// TwinCAT 3 PLC project TcLog
// Title: TcLog
// Company: Benedikt Geisler
// Author: Benedikt Geisler
// ProjectVersion: 0.6.1
// Description: TcLog provides logging functionality to TwinCAT.
// ProgramVersion: 3.1.4026.12
// libraries:
//   Base Interfaces,newest,System
//   Tc2_Standard, * (Beckhoff Automation GmbH)
//   Tc2_System, * (Beckhoff Automation GmbH)
//   Tc2_Utilities, * (Beckhoff Automation GmbH)
//   Tc3_DynamicMemory, * (Beckhoff Automation GmbH)
//   Tc3_Module, * (Beckhoff Automation GmbH)
//   TcUnit, * (www.tcunit.org)
// project tree:
//   / Constants.TcGVL
//   Logger/ LogLevelToAdsLogMsgType.TcPOU, TcLog.TcPOU, TcLogCore.TcPOU, TcLogTrig.TcPOU
//   Logger/_Tests/ TestWrapper_NET.TcPOU
//   StringBuilder/_Interfaces/ ILimitedStringBuilder.TcIO, IStringBuilder.TcIO
//   Utils/ AnyToString.TcPOU, DateTime.TcPOU, DeleteOldFiles.TcPOU, DynamicStringBuffer.TcPOU, GetFileAgeInSeconds.TcPOU
//   Utils/_DataTypes/ DeleteFilesState.TcDUT, PersistToFileState.TcDUT
//   Logger/_DataTypes/ ErrorCodes.TcDUT, LogLevels.TcDUT, RollingIntervals.TcDUT, Error.TcDUT, LoggingConfiguration.TcDUT
//   Logger/_Interfaces/ ILog.TcIO, ILogCore.TcIO
//   StringBuilder/ StringBuilder.TcPOU
//   Utils/_Tests/ ConvertAnyToString_TEST.TcPOU, DateTime_TEST.TcPOU, DynamicStringBuffer_TEST.TcPOU
// real-time tasks:
//   TASK PlcTask1: cycle T#10ms, priority 21, ADS port 351

// ---- Utils/_DataTypes/DeleteFilesState.TcDUT
// States for state machine used in `DeleteOldFiles`.
{attribute 'qualified_only'}
{attribute 'strict'}
TYPE INTERNAL DeleteFilesState :
(
	Idle := 0,
  SearchNextFile,
  WaitUntilExecutionDone,
  ProcessFoundFiles,
  CheckIfFileIsDirectory,
  CheckFileTime,
  DeleteFile,
  FileDeleted
);
END_TYPE

// ---- Utils/_DataTypes/PersistToFileState.TcDUT
// States for state machine used in `DynamicStringBuffer.PersistToFile`
{attribute 'qualified_only'}
{attribute 'strict'}
TYPE INTERNAL PersistToFileState :
(
	Idle := 0,
  OpenFile,
  GetStringFromFifo,
  AppendDataToFile,
  CloseFile
);
END_TYPE

// ---- Logger/_DataTypes/ErrorCodes.TcDUT
/// Provides error codes for TcLogCore
{attribute 'qualified_only'}
{attribute 'strict'}
{attribute 'to_string'}
TYPE ErrorCodes : 
(
	None := 0,
	OpeningFileFailed,
	WritingToFileFailed,
	ClosingFileFailed,
	EnumeratingFilesInSpecifiedDirectoryFailed,
	DeletingFileFailed,
	FifoOverflow
);
END_TYPE

// ---- Logger/_DataTypes/LogLevels.TcDUT
/// Log level of message to be logged.
{attribute 'qualified_only'}
{attribute 'strict'}
{attribute 'to_string'}
TYPE LogLevels :
(
	Debug := 0,
	Information,
	Warning,
	Error,
	Fatal
);
END_TYPE

// ---- Logger/_DataTypes/RollingIntervals.TcDUT
/// Rolling interval to create a new log file when expired. 
{attribute 'qualified_only'}
{attribute 'strict'}
{attrivute 'to_string'}
TYPE RollingIntervals :
(
	None := 0,
	Hourly,
	Daily,
	Monthly
);
END_TYPE

// ---- Logger/_DataTypes/Error.TcDUT
/// This is the error type used in this library.
TYPE Error :
STRUCT
  /// `TRUE` signals an active error
	Active : BOOL;
  /// Error code of type `ErrorCodes`
	Code : INT;
  /// Plain text error message
	Info : Tc2_System.T_MaxString;
END_STRUCT
END_TYPE

// ---- Logger/_DataTypes/LoggingConfiguration.TcDUT
/// Configuration of TcLogCore
TYPE LoggingConfiguration :
STRUCT
  /// File name where the logs should be written to. Should not include path.
	FileName : Tc2_System.T_MaxString;
  /// File path where the logs should be written to. Will be prefixed to `FileName`
	FilePath : Tc2_System.T_MaxString;
  /// Whether to include the instance path of TcLog into the log message or not.
	IncludeInstancePath : BOOL;
  /// Whether to write the logs to ADS output or not.
	WriteToAds : BOOL;
  /// Rolling interval: when to create a new log file.
	RollingInterval : RollingIntervals;
  /// What is the minimum log level that gets logged?
	MinimumLevel : LogLevels;
  /// Which delimiter should be used between the different parts of the log string?
	Delimiter : STRING(1);
  /// When should old log files be deleted? Unit: days. Set it to `0` if log files should never be deleted. 
	LogFileLifespan : UINT;
  /// Format of timestamp. See `TcLogCore.TimestampFormat` for formatting options.
	TimestampFormat : STRING;
  /// Log only valid timestamps (skip log messages during time initialization (first few cycles)
  	ValidTimestampsOnly: BOOL;
END_STRUCT
END_TYPE

// ---- Constants.TcGVL
{attribute 'qualified_only'}
VAR_GLOBAL CONSTANT
  /// Fifo overhead needed to manage the string buffer
  FifoOverhead : UDINT := 10;
  /// Buffer size of temporary buffer used to persist all log messages in one cycle. 
	BufferSize : UDINT := (100 * (Tc2_System.MAX_STRING_LENGTH + FifoOverhead));
END_VAR

// ---- StringBuilder/_Interfaces/ILimitedStringBuilder.TcIO
{attribute 'hide'}
INTERFACE INTERNAL ILimitedStringBuilder

METHOD Append : IStringBuilder // Append text TO t current build STRING.
VAR_INPUT
    Text : Tc2_System.T_MaxString; //Text to append to current build string
END_VAR
END_METHOD

METHOD AppendIf : IStringBuilder
VAR_INPUT
    Condition : BOOL;
    Text : Tc2_System.T_MaxString;
END_VAR
END_METHOD

METHOD Reset : ILimitedStringBuilder //Reset current build STRING TO an empty STRING.
END_METHOD

METHOD ToString : Tc2_System.T_MaxString //Returns current build STRING.
END_METHOD

END_INTERFACE

// ---- StringBuilder/_Interfaces/IStringBuilder.TcIO
{attribute 'hide'}
INTERFACE INTERNAL IStringBuilder

METHOD Append : IStringBuilder // Append text TO t current build STRING.
VAR_INPUT
    Text : Tc2_System.T_MaxString; //Text to append to current build string
END_VAR
END_METHOD

METHOD AppendIf : IStringBuilder
VAR_INPUT
    Condition : BOOL;
    Text : Tc2_System.T_MaxString;
END_VAR
END_METHOD

METHOD InsertAtLocation : IStringBuilder
VAR_INPUT
    Text : Tc2_System.T_MaxString;
    Position : INT;
END_VAR
END_METHOD

METHOD PadLeft : IStringBuilder
VAR_INPUT
    text : Tc2_System.T_MaxString; // Text to append to current build string
    length : INT; // Total length of text + padding
    c : STRING(1); // Character to be padded left of text
END_VAR
END_METHOD

METHOD Reset : ILimitedStringBuilder //Reset current build STRING TO an empty STRING.
END_METHOD

METHOD ToString : Tc2_System.T_MaxString //Returns current build STRING.
END_METHOD

END_INTERFACE

// ---- Logger/_Interfaces/ILog.TcIO
INTERFACE ILog

METHOD SetLogger : BOOL
VAR_INPUT
    ref2Core : ILogCore;
END_VAR
END_METHOD

END_INTERFACE

// ---- Logger/_Interfaces/ILogCore.TcIO
INTERFACE ILogCore EXTENDS __System.IQueryInterface

// Logger method.
// Logs data in custom format. No additional formatting will be done.
METHOD LogCustomFormat : BOOL
VAR_INPUT
    data : Tc2_System.T_MaxString; // Data to be logged. No additional formatting will be done.
END_VAR
END_METHOD

// Logger method.
// Logs in the standard format. This includes
// - timestamp
// - log level
// - log message
// - instance path of logging source (optional)
// The message will only be logged if the logging level exceeds the configured minimum logging level.
METHOD LogStandardFormat : BOOL
VAR_INPUT
    data : Tc2_System.T_MaxString; // Data to be logged. Additional formatting wil be done.
    instancePath : Tc2_System.T_MaxString; // Instance path of calling logger to locate source of logging message.
    logLevel : LogLevels; // Log level of message.
END_VAR
END_METHOD

END_INTERFACE

// ---- Logger/LogLevelToAdsLogMsgType.TcPOU
// Converts TcLog.LogLevels into Tc2_System.ADSLOG_MSGTYPEs.
{attribute 'hide'}
FUNCTION INTERNAL LogLevelToAdsLogMsgType : DWORD
VAR_INPUT
  logLevel : LogLevels;
END_VAR
VAR
  _retVal : DWORD;
END_VAR

CASE logLevel OF
  LogLevels.Debug, LogLevels.Information:
    _retVal := Tc2_System.ADSLOG_MSGTYPE_HINT;
  LogLevels.Warning:
    _retVal := Tc2_System.ADSLOG_MSGTYPE_WARN;
  LogLevels.Error, LogLevels.Fatal:
    _retVal := Tc2_System.ADSLOG_MSGTYPE_ERROR;
  ELSE
    _retVal := Tc2_System.ADSLOG_MSGTYPE_HINT;
END_CASE

LogLevelToAdsLogMsgType := _retVal;

END_FUNCTION

// ---- Logger/TcLog.TcPOU
/// `TcLog` is the client side of the logger.  
///
/// It is used to send the logs to `TcLogCore`. Typically, it is instantiated
/// once in each `FUNCTION_BLOCK` or `PROGRAM` where logging is done. The same 
/// instance can then be used for all logging within that POU. 
///
/// `TcLog` implements a string builder that facilitates the compilation of the log
/// message without the need for external data type conversions or multiple chained `CONCAT` calls.
/// See the method section for more information.
///
/// The last method to call after the log message has been built is one of ´[Debug|Information|Warning|Error|Fatal]`. 
/// This sets the log level of the message and sends it off to the log message queue of `TcLogCore` where it will
/// be processed according to its configuration.
{attribute 'hide_all_locals'}
{attribute 'reflection'} 
FUNCTION_BLOCK TcLog IMPLEMENTS ILog
VAR
  _logConditionSatisfied : BOOL; // flag that indicates, whether log condition has been satisfied.
                                // Logging will only be carried out it this evaluates to TRUE.                    
  _logDataInitialized : BOOL; // flag that indicate, whether log data has been initialized.
                             // Necessary for configuration methods to provide a fluent interface.                            
  _logData : Tc2_System.T_MaxString; // contains message to be logged.
  _usedLogger : ILogCore;
  {attribute 'instance-path'} 
  {attribute 'noinit'} 
  _instancePath : STRING; // contains instance path
END_VAR
VAR_STAT
  {attribute 'hide'}
  s_loggerSingletonInstance : ILogCore; // Wires up TcLog ("Client") to TcLogCore ("Server") (Singleton-Behaviour)
END_VAR
VAR CONSTANT
  InvalidLoggerReference : UDINT := 0;
END_VAR

/// Appends any given data to the log string. The type of the provided data
/// has to be one of the [standard data types](https://infosys.beckhoff.com/english.php?content=../content/1033/tc3_plc_intro/2529388939.html&id=).
/// This method can be chained.
METHOD AppendAny : REFERENCE TO TcLog
VAR_INPUT
  /// data to be appended to log string.
  data : ANY;
END_VAR
InitializeLogData();

_logData := Tc2_Standard.CONCAT(_logData, AnyToString(data));

AppendAny REF= THIS^;
END_METHOD

/// Appends another string to the log message.
/// This method can be chained.
METHOD AppendString : REFERENCE TO TcLog
VAR_INPUT
  /// data to be appended to log string.
  data : Tc2_System.T_MaxString; 
END_VAR
InitializeLogData();

_logData := Tc2_Standard.CONCAT(_logData, data);
  
AppendString REF= THIS^;
END_METHOD

/// Appends information about the given variable to the log string. 
/// This method can be chained.
/// Example: 

/// ```st
/// VAR
///   Logger: TcLog;
///    myInt : INT := 10;
///   myVarInfo : __SYSTEM.VAR_INFO := __VARINFO(myInt);
/// END_VAR
/// Logger.AppendVariable(myVarInfo, myInt);
/// ```
///
METHOD AppendVariable : REFERENCE TO TcLog
VAR_INPUT
  /// [VAR_INFO](https://infosys.beckhoff.com/index.php?content=../content/1031/tc3_plc_intro/3527777675.html&id=) of variable to be appended to log string.
  varInfo : __SYSTEM.VAR_INFO;
  /// Value of variable to be appended to log string.
  value : ANY; 
END_VAR
VAR
  format : Tc2_Utilities.FB_FormatString;
  symbolName : Tc2_System.T_MaxString;
  typeName : Tc2_System.T_MaxString;
END_VAR
InitializeLogData();

symbolName := varInfo.Symbol;
typeName := varInfo.TypeName; 

format(
  sFormat := '%s [%s] : ',
  arg1 := Tc2_Utilities.F_STRING(symbolName),
  arg2 := Tc2_Utilities.F_STRING(typeName));
  
AppendString(format.sOut);
AppendAny(value);

AppendVariable REF= THIS^;
END_METHOD

/// Logs the log string in DEBUG level.
METHOD Debug : BOOL
VAR_INPUT
  /// Message to be appended to log string.
  message : Tc2_System.T_MaxString; 
END_VAR
InitializeLogData();
IF _logConditionSatisfied THEN
  IF _usedLogger <> InvalidLoggerReference THEN 
    _usedLogger.LogStandardFormat(Tc2_Standard.CONCAT(_logData, message), ShortenInstancePath(_instancePath), LogLevels.Debug); 
  ELSE
    Tc2_System.ADSLOGSTR(ADSLOG_MSGTYPE_LOG OR LogLevelToAdsLogMsgType(LogLevels.Error), 'usedLogger: No valid reference', ''); 
  END_IF
END_IF
_logDataInitialized := FALSE;
END_METHOD

/// Logs the log string in ERROR level.
METHOD Error : BOOL
VAR_INPUT
  /// Message to be appended to log string.
  message : Tc2_System.T_MaxString; 
END_VAR
InitializeLogData();
IF _logConditionSatisfied THEN
  IF _usedLogger <> InvalidLoggerReference THEN 
    _usedLogger.LogStandardFormat(Tc2_Standard.CONCAT(_logData, message), ShortenInstancePath(_instancePath), LogLevels.Error); 
  ELSE
    Tc2_System.ADSLOGSTR(ADSLOG_MSGTYPE_LOG OR LogLevelToAdsLogMsgType(LogLevels.Error), 'usedLogger: No valid reference', ''); 
  END_IF
END_IF
_logDataInitialized := FALSE;
END_METHOD

/// Logs the log string in FATAL level.
METHOD Fatal : BOOL
VAR_INPUT
  /// Message to be appended to log string.
  message : Tc2_System.T_MaxString; 
END_VAR
InitializeLogData();
IF _logConditionSatisfied THEN
  IF _usedLogger <> InvalidLoggerReference THEN 
    _usedLogger.LogStandardFormat(Tc2_Standard.CONCAT(_logData, message), ShortenInstancePath(_instancePath), LogLevels.Fatal); 
  ELSE
    Tc2_System.ADSLOGSTR(ADSLOG_MSGTYPE_LOG OR LogLevelToAdsLogMsgType(LogLevels.Error), 'usedLogger: No valid reference', ''); 
  END_IF
END_IF
_logDataInitialized := FALSE;
END_METHOD

/// Logs the log string in INFORMATION level.
METHOD Information : BOOL
VAR_INPUT
  /// Message to be appended to log string.
  message : Tc2_System.T_MaxString; 
END_VAR
InitializeLogData();
IF _logConditionSatisfied THEN
  IF _usedLogger <> InvalidLoggerReference THEN 
    _usedLogger.LogStandardFormat(Tc2_Standard.CONCAT(_logData, message), ShortenInstancePath(_instancePath), LogLevels.Information); 
  ELSE
    Tc2_System.ADSLOGSTR(ADSLOG_MSGTYPE_LOG OR LogLevelToAdsLogMsgType(LogLevels.Error), 'usedLogger: No valid reference', ''); 
  END_IF
END_IF
_logDataInitialized := FALSE;
END_METHOD

/// Initializes the reference to the core logger. Should only be called once from the core logger directly.
METHOD PUBLIC Init : BOOL
VAR_INPUT
  /// Reference to TcLoggerCore instance.
  ref2Core : ILogCore; 
END_VAR
IF s_loggerSingletonInstance = 0 THEN
	s_loggerSingletonInstance := ref2Core;
END_IF
END_METHOD

// Necessary to provide a fluent interface of the function. 
// Has to be called at the begin of any method that returns a reference to THIS^
METHOD PRIVATE InitializeLogData : BOOL
IF NOT _logDataInitialized THEN
  _logConditionSatisfied := TRUE;
  _logData := '';
  _logDataInitialized := TRUE;
  IF _usedLogger = 0 THEN _usedLogger := s_loggerSingletonInstance; END_IF
END_IF
END_METHOD

/// Conditional execution of the log command. Only executes logging when Cond = TRUE.
METHOD OnCondition : REFERENCE TO TcLog
VAR_INPUT
  /// Logs data only if this condition evaluates to TRUE.
  cond : BOOL; 
END_VAR
InitializeLogData();

_logConditionSatisfied := cond;

OnCondition REF= THIS^;
END_METHOD

/// Initializes the reference to the core logger. This enables you to use several
/// loggers with different configurations in one project.
METHOD SetLogger : BOOL
VAR_INPUT
  /// Reference to Core Logger
  ref2Core : ILogCore; 
END_VAR
_usedLogger := ref2Core;
END_METHOD

// Helper method. Shortens the instance path by omitting superfluent information
// such as concrete logger instance and plc/project names.
{attribute 'hide'}
METHOD PRIVATE ShortenInstancePath : Tc2_System.T_MaxString
VAR_INPUT
  path : Tc2_System.T_MaxString; // Instance path to be shortened.
END_VAR
VAR
  i : UINT;
  shortenedPath : Tc2_System.T_MaxString;
  positionInString : INT := 0;
  positionOfLastDot : INT := 0;
END_VAR
shortenedPath := path;

// Find last '.'
WHILE(Tc2_Standard.FIND(shortenedPath, '.') > 0) DO
  positionInString := Tc2_Standard.FIND(shortenedPath, '.');
  shortenedPath := Tc2_Standard.DELETE(shortenedPath, positionInString+1, 0); 
  positionOfLastDot := positionOfLastDot+positionInString;
END_WHILE

shortenedPath := Path;
// Delete instantiation of this FB (obvious information)
shortenedPath := Tc2_Standard.DELETE(shortenedPath, Tc2_Standard.LEN(shortenedPath)-positionOfLastDot+1, positionOfLastDot);
// Delete project information
positionInString := Tc2_Standard.FIND(shortenedPath, '.');
shortenedPath := Tc2_Standard.DELETE(shortenedPath, positionInString+1, 0);
// Delete PLC information
positionInString := Tc2_Standard.FIND(shortenedPath, '.');
shortenedPath := Tc2_Standard.DELETE(shortenedPath, positionInString+1, 0);

ShortenInstancePath := shortenedPath;
END_METHOD

/// Logs directly to ADS log, ignoring the settings of the base logger.
METHOD ToAdsLog : BOOL
VAR_INPUT
  /// Log level in which message should be logged to ADS.
  logLevel : LogLevels; 
END_VAR
InitializeLogData();

IF _logConditionSatisfied THEN
  Tc2_System.ADSLOGSTR(ADSLOG_MSGTYPE_LOG OR LogLevelToAdsLogMsgType(logLevel), _logData, ''); 
END_IF

_logDataInitialized := FALSE;
END_METHOD

/// Saves custom formatted log string. 
/// No addtitional information will be added, no formatting will be applied.
METHOD ToCustomFormat : BOOL
VAR_INPUT
  /// Message to be appended to log string.
  message : Tc2_System.T_MaxString; 
END_VAR
InitializeLogData();
IF _logConditionSatisfied THEN
  IF _usedLogger <> InvalidLoggerReference THEN 
    _usedLogger.LogCustomFormat(Tc2_Standard.CONCAT(_logData, message)); 
  ELSE
    Tc2_System.ADSLOGSTR(ADSLOG_MSGTYPE_LOG OR LogLevelToAdsLogMsgType(LogLevels.Error), 'usedLogger: No valid reference', ''); 
  END_IF
END_IF
_logDataInitialized := FALSE;
END_METHOD

/// Logs the log string in WARNING level.
METHOD Warning : BOOL
VAR_INPUT
  /// Message to be appended to log string.
  message : Tc2_System.T_MaxString; 
END_VAR
InitializeLogData();
IF _logConditionSatisfied THEN
  IF _usedLogger <> InvalidLoggerReference THEN 
    _usedLogger.LogStandardFormat(Tc2_Standard.CONCAT(_logData, message), ShortenInstancePath(_instancePath), LogLevels.Warning); 
  ELSE
    Tc2_System.ADSLOGSTR(ADSLOG_MSGTYPE_LOG OR LogLevelToAdsLogMsgType(LogLevels.Error), 'usedLogger: No valid reference', ''); 
  END_IF
END_IF
_logDataInitialized := FALSE;
END_METHOD

END_FUNCTION_BLOCK

// ---- Utils/AnyToString.TcPOU
/// Converts value of input data to string, where the input type can be any of 
/// the standard data types.
FUNCTION AnyToString : Tc2_System.T_MaxString
VAR_INPUT
  /// Input data
  data : ANY;
END_VAR
VAR
  _anyByte : POINTER TO BYTE;
  _anyUSINT : POINTER TO USINT;
  _anyInt : POINTER TO INT;
  _anyUInt : POINTER TO UINT;
  _anyUDInt : POINTER TO UDINT;
  _anySInt : POINTER TO SINT;
  _anyDInt : POINTER TO DINT;
  _anyLInt : POINTER TO LINT;
  _anyULInt : POINTER TO ULINT;
  _anyWord : POINTER TO WORD;
  _anyLWord : POINTER TO LWORD;
  _anyReal : POINTER TO REAL;
  _anyLReal : POINTER TO LREAL;
  _anyDateAndTime : POINTER TO DATE_AND_TIME;
  _anyDate : POINTER TO DATE;
  _anyTime : POINTER TO TIME;
  _anyWString : POINTER TO WSTRING;
  _anyTOD : POINTER TO TOD;
  _anyString : POINTER TO STRING;
  _string : T_MAXSTRING;
  _wString : WSTRING;
END_VAR

IF data.TypeClass = __SYSTEM.TYPE_CLASS.TYPE_BYTE THEN
  _anyByte := data.pValue;
  AnyToString := BYTE_TO_STRING(_anyByte^);
    
ELSIF data.TypeClass = __SYSTEM.TYPE_CLASS.TYPE_INT THEN
  _anyInt := data.pValue;
  AnyToString := INT_TO_STRING(_anyInt^);
    
ELSIF data.TypeClass = __SYSTEM.TYPE_CLASS.TYPE_UINT THEN
  _anyUInt := data.pValue;
  AnyToString := UINT_TO_STRING(_anyUInt^);
    
ELSIF data.TypeClass = __SYSTEM.TYPE_CLASS.TYPE_UDINT THEN
  _anyUDInt := data.pValue;
  AnyToString := UDINT_TO_STRING(_anyUDInt^);
    
ELSIF data.TypeClass = __SYSTEM.TYPE_CLASS.TYPE_SINT THEN
  _anySInt := data.pValue;
  AnyToString := SINT_TO_STRING(_anySInt^);
    
ELSIF data.TypeClass = __SYSTEM.TYPE_CLASS.TYPE_USINT THEN
  _anyUSInt := data.pValue;
  AnyToString := USINT_TO_STRING(_anyUSInt^);
    
ELSIF data.TypeClass = __SYSTEM.TYPE_CLASS.TYPE_DINT THEN
  _anyDInt := data.pValue;
  AnyToString := DINT_TO_STRING(_anyDInt^);
    
ELSIF data.TypeClass = __SYSTEM.TYPE_CLASS.TYPE_LINT THEN
  _anyLInt := data.pValue;
  AnyToString := LINT_TO_STRING(_anyLInt^);
      
ELSIF data.TypeClass = __SYSTEM.TYPE_CLASS.TYPE_ULINT THEN
  _anyULInt := data.pValue;
  AnyToString := ULINT_TO_STRING(_anyULInt^);
  
ELSIF data.TypeClass = __SYSTEM.TYPE_CLASS.TYPE_WORD THEN
  _anyWord := data.pValue;
  AnyToString := WORD_TO_STRING(_anyWord^);
    
ELSIF data.TypeClass = __SYSTEM.TYPE_CLASS.TYPE_LWORD THEN
  _anyLWord := data.pValue;
  AnyToString := LWORD_TO_STRING(_anyLWord^);
  
ELSIF data.TypeClass = __SYSTEM.TYPE_CLASS.TYPE_REAL THEN
  _anyReal := data.pValue;
  AnyToString := REAL_TO_STRING(_anyReal^);
  
ELSIF data.TypeClass = __SYSTEM.TYPE_CLASS.TYPE_LREAL THEN
  _anyLReal := data.pValue;
  AnyToString := LREAL_TO_STRING(_anyLReal^);
  
ELSIF data.TypeClass = __SYSTEM.TYPE_CLASS.TYPE_DATEANDTIME THEN
  _anyDateAndTime := data.pValue;
  AnyToString := DT_TO_STRING(_anyDateAndTime^);  
  
ELSIF data.TypeClass = __SYSTEM.TYPE_CLASS.TYPE_DATE THEN
  _anyDate := data.pValue;
  AnyToString := DATE_TO_STRING(_anyDate^);
  
ELSIF data.TypeClass = __SYSTEM.TYPE_CLASS.TYPE_TIME THEN
  _anyTime := data.pValue;
  AnyToString := TIME_TO_STRING(_anyTime^);
  
ELSIF data.TypeClass = __SYSTEM.TYPE_CLASS.TYPE_STRING THEN
  _anyString := data.pValue;
  AnyToString := _anyString^;
  
ELSIF data.TypeClass = __SYSTEM.TYPE_CLASS.TYPE_WSTRING THEN
  _anyWString := data.pValue;
  _wString := _anyWString^;
  Tc2_Utilities.WSTRING_TO_STRING2(ADR(_string), ADR(_wString), SIZEOF(_wString));
  AnyToString := _string;
  
ELSIF data.TypeClass = __SYSTEM.TYPE_CLASS.TYPE_TIMEOFDAY THEN
  _anyTOD := data.pValue;
  AnyToString := TOD_TO_STRING(_anyTOD^);
  
ELSE
  AnyToString := TO_STRING(data.pValue^);
END_IF

END_FUNCTION

// ---- Logger/TcLogCore.TcPOU
/// `TcLogCore` provides the base functionality of the logger and sets the configuration.
/// The logger can be configured by calling its methods that set the configuration.
///
/// > [!NOTE]
/// > `TcLogCore.RunLogger()` should be called once each cycle. The configuration methods should be called **before** 
/// > `RunLogger` is called.
///
/// When declaring an instance of TcLogCore, the ininital buffer size has to be set. If the buffer size is set too low, it will expand
/// automatically if enough memory is available.
///
/// To set the inital buffer size to accomodate 100 messages, use it like this:
///
/// ```st
/// VAR
///   myLogger: TcLogCore(BufferSize := 100 * (Tc2_System.MAX_STRING_LENGTH * Constants.FifoOverhead));
/// END_VAR
/// ```
///
{attribute 'hide_all_locals'}
FUNCTION_BLOCK TcLogCore IMPLEMENTS ILogCore
VAR
	_loggingSingleton : TcLog; // Logger-Singleton: Required to provide Singleton-functionality for TcLog.
	_utcTimeAsFileTime : Tc2_Utilities.T_FILETIME; // Current utc time as filetime
	_localTimeAsSystemTime : Tc2_Utilities.TIMESTRUCT; // Current local time as timestring
	_localTimeAsString : STRING; // Current local time as string
	_logCache : DynamicStringBuffer; // Dynamic string buffer to cache logs to be processed
	_startLoggingConfiguration : BOOL; // Aux variable to provide fluent interface.
	_internalErrorOccured : BOOL; // Aux variable to log internal errors to Error-property.                                                   				
	_config : LoggingConfiguration; // Logging configuration. Is set by invoking configuration methods.
	_error : Error; // Contains information about internal error.
	_busy : BOOL; // Logger is busy, typically with writing logs to the file system.
  _timeInfoReady : BOOL := FALSE; // Set to true once the time information is available
END_VAR

// Nothing to be done here. Logger works by invoking its methods.
// "RunLogger" contains all the implementation that has to be processed cyclically.

// Builds logging configuration.
// Required to provide a fluent interface.
// Has to be called at the begin of each method that configures the logger.
{attribute 'hide'}
METHOD PRIVATE BuildLoggingConfiguration : BOOL
IF NOT _startLoggingConfiguration THEN
	_startLoggingConfiguration := TRUE;
	
	_config.RollingInterval := RollingIntervals.Daily;
	_config.WriteToAds := FALSE;
	_config.FileName := '';
	_config.FilePath := 'c:\';
	_config.MinimumLevel := LogLevels.Debug;
	_config.Delimiter := '|';
	_config.IncludeInstancePath := FALSE;
	_config.LogFileLifespan := 0;
	_config.TimestampFormat := 'YYYYMMDD_hhmm_';
	_config.ValidTimestampsOnly := FALSE;
END_IF
END_METHOD

/// `Busy` evaluates to `TRUE` as long as the log file is kept open to append new log messages
/// or there are pending messages in the queue to be written to the logfile.
{attribute 'monitoring':='call'}
PROPERTY Busy : BOOL
GET
Busy := _busy;
END_GET
SET // PRIVATE
_busy := Busy;
END_SET
END_PROPERTY

/// Returns the current configuration of the logger.
{attribute 'monitoring':='variable'}
PROPERTY Configuration : LoggingConfiguration
GET
Configuration := _config;
END_GET
END_PROPERTY

/// Configuration method which sets the lifespan of log files. Once exceeded, they will be deleted.
METHOD DeleteLogFilesAfterDays : REFERENCE TO TcLogCore
VAR_INPUT
  /// Lifespan of logfiles in days.
	lifespan : UINT; 
END_VAR
BuildLoggingConfiguration();

_config.LogFileLifespan := lifespan;

DeleteLogFilesAfterDays REF= THIS^;
END_METHOD

/// Returns information about internal errors.
{attribute 'monitoring':='call'}
PROPERTY Error : REFERENCE TO Error
GET
Error REF= _error;
END_GET
END_PROPERTY

METHOD FB_init : BOOL
VAR_INPUT
	bInitRetains : BOOL; // if TRUE, the retain variables are initialized (warm start / cold start)
	bInCopyCode : BOOL; // if TRUE, the instance afterwards gets moved into the copy code (online change)
  /// Initial buffer size for the internal log message buffer
	bufferSize : UDINT;
END_VAR
_loggingSingleton.Init(THIS^);
_logCache.Init(bufferSize);
END_METHOD

/// Flushes the logging cache. All messages that have not yet been processed will be lost.
METHOD FlushCache : BOOL
_logCache.FlushCache();
END_METHOD

/// Configuration method. If this method is called, the instance path where the log 
/// messages has been triggered will be included in the log message. 
METHOD IncludeInstancePath : REFERENCE TO TcLogCore
BuildLoggingConfiguration();

_config.IncludeInstancePath := TRUE;

IncludeInstancePath REF= This^;
END_METHOD

/// Logger method. It should only be called from within objects that implement `ILog`.
/// Logs data in custom format. No additional formatting will be done. 
METHOD LogCustomFormat : BOOL
VAR_INPUT
  /// Data to be logged.
	data : Tc2_System.T_MaxString; 
END_VAR
IF(TimeInfoReady OR NOT _config.ValidTimestampsOnly) THEN 
	IF _config.WriteToAds THEN 
		Tc2_System.ADSLOGSTR(ADSLOG_MSGTYPE_LOG OR ADSLOG_MSGTYPE_HINT, data, ''); 
	END_IF
	
	IF _config.FileName <> '' THEN 
		_logCache.AddLine(data);
	END_IF
END_IF
END_METHOD

/// Logger method. It should only be called from within objects that implement `ILog`.
/// Logs in the standard format. This includes
/// - timestamp
/// - log level
/// - log message
/// - instance path of logging source (optional)
/// The message will only be logged if the logging level exceeds the configured minimum logging level.
METHOD LogStandardFormat : BOOL
VAR_INPUT
  /// Data to be logged.
	data : Tc2_System.T_MaxString; 
  /// Instance path of calling logger to locate source of logging message.
	instancePath : Tc2_System.T_MaxString;
  /// Log level of message. 
	logLevel : LogLevels; 
END_VAR
VAR_INST
  {attribute 'hide'}
	messageBuilder : StringBuilder;
END_VAR
IF LogLevel >= _config.MinimumLevel AND (TimeInfoReady OR NOT _config.ValidTimestampsOnly)  THEN
	IF _config.WriteToAds THEN 
		Tc2_System.ADSLOGSTR(
			ADSLOG_MSGTYPE_LOG OR LogLevelToAdsLogMsgType(logLevel), 
			messageBuilder
				.Reset()
				.AppendIf(_config.IncludeInstancePath, instancePath)
				.AppendIf(_config.IncludeInstancePath, _config.Delimiter)
				.Append(data)
				.ToString(), 
			''
		); 
	END_IF
	
	IF _config.FileName <> '' THEN 
		_logCache.AddLine(
			messageBuilder
					.Reset()
					.Append(_localTimeAsString)
					.Append(_config.Delimiter)
					.Append(TO_STRING(LogLevel))
					.AppendIf(_config.IncludeInstancePath, _config.Delimiter)
					.AppendIf(_config.IncludeInstancePath, instancePath)
					.Append(_config.Delimiter)
					.Append(data)
					.ToString()
		);
	END_IF
END_IF
END_METHOD

/// Configuration method.
/// Sets the minimum log level. Log messages below this level 
/// will not be logged.
METHOD MinimumLevel : REFERENCE TO TcLogCore
VAR_INPUT
  /// Minimum log level to be logged.
	level : LogLevels; 
END_VAR
BuildLoggingConfiguration();

_config.MinimumLevel := level;

MinimumLevel REF=THIS^;
END_METHOD

// Checks the specified rolling interval for the file name.
// Generates new file name if rolling intervall exceeded.
{attribute 'hide_all_locals'}
{attribute 'hide'}
METHOD PRIVATE RollingIntervalReached : BOOL
VAR_INPUT
	currentUtcTime : Tc2_Utilities.TIMESTRUCT;  // Current system time as utc
	rollingInterval : RollingIntervals; // Rolling interval 
END_VAR
VAR_INST
	newHour : Tc2_Standard.R_TRIG;
	newDay : Tc2_Standard.R_TRIG;
	newMonth : Tc2_Standard.R_TRIG;
	
	hourRolled : BOOL;
	dayRolled : BOOL;
	monthRolled : BOOL;
END_VAR
newHour(CLK := (currentUtcTime.wMinute = 0 AND currentUtcTime.wSecond = 0), 
	Q => hourRolled);
newDay(CLK := (hourRolled AND currentUtcTime.wHour = 0), 
	Q => dayRolled);
newMonth(CLK := (dayRolled AND currentUtcTime.wDay = 1), 
	Q => monthRolled);

RollingIntervalReached := 	(hourRolled 	AND rollingInterval = RollingIntervals.Hourly) OR
							(dayRolled 		AND rollingInterval = RollingIntervals.Daily) 	OR
							(monthRolled 	AND rollingInterval = RollingIntervals.Monthly);
END_METHOD

/// Cyclic method of Logger.
/// This method has to be executed in every plc cycle and runs 
/// all internal methods that have to be executed cyclically.
/// > [!NOTE]
/// > This method should be the last method of `TcLogCore` to be called in each cycle.
{attribute 'hide_all_locals'}
METHOD RunLogger : BOOL
VAR_INST
	newDay : Tc2_Standard.R_TRIG; 
	dateTime : DateTime;
	deleteExpiredLogFiles : DeleteOldFiles;
	fileNameStringBuilder : StringBuilder;
	timeStamp : STRING; // Timestamp used for filename
END_VAR
// Generate time data (shared state)
dateTime();
IF dateTime.Done THEN _timeInfoReady := TRUE; END_IF

_localTimeAsSystemTime := dateTime.AsLocalSystemTime;
_localTimeAsString := dateTime.AsLocalSystemTimeString;
_utcTimeAsFileTime := dateTime.AsUtcFileTime;

// Generate new timestamp for filename
IF RollingIntervalReached(_localTimeAsSystemTime, _config.RollingInterval) OR dateTime.Done THEN
	timeStamp := dateTime.ToFormatString(_config.TimestampFormat);
END_IF

// Delete expired log files
newDay(CLK := _localTimeAsSystemTime.wHour = 0);
deleteExpiredLogFiles(
	StartScan 			:= 	newDay.Q AND (_config.LogFileLifespan > 0),
	ExpirationInDays 	:=	_config.LogFileLifespan,
	FilePath			:=	_config.FilePath,
	FileName 			:=	_config.FileName,
	CurrentUtcTime 		:= 	_utcTimeAsFileTime	
	);
IF deleteExpiredLogFiles.Error.Active THEN
	_internalErrorOccured := TRUE;
	_error := deleteExpiredLogFiles.Error;
END_IF
		
// Persist logging messages to file
_logCache.PersistToFile(
  TimeInfoReady,
	fileNameStringBuilder
		.Reset()
		.Append(_config.FilePath)
		.AppendIf(Tc2_Standard.RIGHT(_config.FilePath, 1) <> '\', '\')
		.Append(timeStamp)
		.Append(_config.FileName)
		.ToString()
);
IF _logCache.Error.Active THEN
	_internalErrorOccured := TRUE;
	_error := _logCache.Error;
END_IF

// Forward busy state of LogCache 
Busy := _logCache.Busy;

// Reset Logging configuration: neccesary in order to provide fluent interface
_startLoggingConfiguration := FALSE;

// Reset error flag each cycle to automatically confirm errors once they are gone.
IF NOT _internalErrorOccured THEN
	_error.Active := FALSE;
	_error.Code := ErrorCodes.None;
	_error.Info := '';
END_IF
_internalErrorOccured := FALSE;
END_METHOD

/// Configuration method
/// Sets delimiter between different columns of log file.
METHOD SetDelimiter : REFERENCE TO TcLogCore
VAR_INPUT
  /// Delimiter between different columns of log file.
	delimiter : STRING(1); 
END_VAR
BuildLoggingConfiguration();

_config.Delimiter := delimiter;

SetDelimiter REF=THIS^;
END_METHOD

/// Configuration method.
/// Sets the rolling interval of the log file. Once the rolling interval
/// expires, a file name with a new timestamp will be generated.
METHOD SetRollingInterval : REFERENCE TO TcLogCore
VAR_INPUT
  /// Rolling interval for log file. Once exceeded, a new log file will be created.
	interval : RollingIntervals; 
END_VAR
BuildLoggingConfiguration();

_config.RollingInterval := interval;

SetRollingInterval REF= THIS^;
END_METHOD

/// `TimeInfoReady` evaluates to `TRUE` once the time information used by determine
/// the timestamp for the message is available.
{attribute 'monitoring':='call'}
PROPERTY TimeInfoReady : BOOL
GET
TimeInfoReady := _timeInfoReady;
END_GET
END_PROPERTY

/// Configuration method.
/// Sets the format of the timestamp in the file name. 
/// 
/// The following format options are available:
///	Y : year
///	M : month
/// D : day
/// h : hour 
/// m : minute
/// s : second
/// i : millisecond
/// 
/// Example: _YYMMDD-hh:mm:ss:iii_
/// => _20210812-12:30:22:123_
METHOD TimestampFormat : REFERENCE TO TcLogCore
VAR_INPUT
  /// Format the timestamp should have.
	format : STRING; 
END_VAR
BuildLoggingConfiguration();

_config.TimestampFormat := format;

TimestampFormat REF= THIS^;
END_METHOD

/// Configuration method. If this method is called, only valid timestamps are logged.
/// Note that using this configuration will skip logging anything during the first few PLC cycles, 
/// as TwinCAT needs a few cycles to initialize its time information.
METHOD ValidTimestampsOnly : REFERENCE TO TcLogCore
BuildLoggingConfiguration();

_config.ValidTimestampsOnly := TRUE;

ValidTimestampsOnly REF= This^;
END_METHOD

/// Configuration method.
/// If this method is called, the logs will be written to ADS.
METHOD WriteToAds : REFERENCE TO TcLogCore
BuildLoggingConfiguration();

_config.WriteToAds := TRUE;

WriteToAds REF= This^;
END_METHOD

/// Configuration method.
/// If this method is called, the logs will be persisted to the file system.
METHOD WriteToFile : REFERENCE TO TcLogCore
VAR_INPUT
  /// File path the logs will be written to.
	path : Tc2_System.T_MaxString; 
  /// File name of the log file. Will automatically be prefixed by timestamp.
	fileName : STRING; 
END_VAR
BuildLoggingConfiguration();

IF Tc2_Standard.RIGHT(path, 1) <> '\' THEN
  _config.FilePath := TC2_Standard.CONCAT(path, '\');  
ELSE
  _config.FilePath := path;
END_IF
_config.FileName := fileName;

WriteToFile REF= This^;
END_METHOD

END_FUNCTION_BLOCK

// ---- Utils/DynamicStringBuffer.TcPOU
{attribute 'hide_all_locals'}
FUNCTION_BLOCK INTERNAL DynamicStringBuffer
VAR_OUTPUT
  Error : Error; // Error information of this FB
END_VAR
VAR
  _fifo : Tc2_Utilities.FB_StringRingBuffer; // Necessary to buffer log data until it has been written to file.
  _memoryManager : Tc3_DynamicMemory.FB_DynMem_Manager; // Memory manager, required by DynMem_Buffer.
  _dynamicMemoryBuffer : Tc3_DynamicMemory.FB_DynMem_Buffer(ipMemMan := _memoryManager); // Provides dynamic buffer for Fifo. Is extended automatically if more than the
                                                                   // default buffer size is needed.                  
  _busy : BOOL; // Buffer is busy; typically with writing data to the file system.
END_VAR

METHOD AddLine : BOOL
VAR_INPUT
  text : Tc2_System.T_MaxString; // Text to be added to the buffer
END_VAR
ResizeFifoBufferIfNecessary();
_fifo.A_AddTail(putValue := Tc2_Standard.CONCAT(Tc2_Standard.LEFT(text, 254), '$N'));
END_METHOD

METHOD AddString : BOOL
VAR_INPUT
  text : Tc2_System.T_MaxString; // String to be added to the buffer
END_VAR
ResizeFifoBufferIfNecessary();
_fifo.A_AddTail(putValue := text);
END_METHOD

METHOD PRIVATE AllocateBuffer : BOOL // Allocates buffer FOR the fifo.
VAR_INPUT
  bufferSize : UDINT; // Initial buffer size in BYTEs for fifo buffer.
END_VAR
_dynamicMemoryBuffer.CreateBuffer(nSize:=bufferSize, bReset:=TRUE);
_fifo.pBuffer := _dynamicMemoryBuffer.pBuffer;
_fifo.cbBuffer := bufferSize;
END_METHOD

{attribute 'monitoring':='call'}
PROPERTY Busy : BOOL
GET
Busy := _busy;
END_GET
SET // PRIVATE
_busy := Busy;
END_SET
END_PROPERTY

METHOD FB_exit : BOOL
VAR_INPUT
  bInCopyCode : BOOL; // if TRUE, the exit method is called for exiting an instance that is copied afterwards (online change).
END_VAR
_dynamicMemoryBuffer.Clear();
END_METHOD

METHOD FlushCache : BOOL
_fifo.A_Reset();
END_METHOD

METHOD INTERNAL Init : BOOL
VAR_INPUT
  bufferSize : UDINT; // Initial buffer size in BYTEs for fifo buffer.
END_VAR
AllocateBuffer(bufferSize);
END_METHOD

{attribute 'hide_all_locals'}
METHOD PersistToFile : BOOL
VAR_INPUT
  enable: BOOL; // TRUE starts persistence mechanism
  fileName : Tc2_System.T_MaxString; // File name including its path
END_VAR
VAR_INST
  state : PersistToFileState;
  
  fileOpen : Tc2_System.FB_FileOpen;
  fileHandle : UINT;
  
  fileWrite : Tc2_System.FB_FileWrite;
  lockFileWriteToForceRisingEdge : BOOL; // filePuts can only be executed every other cycle
                                         // since it needs a rising edge to execute.
  fileClose : Tc2_System.FB_FileClose;
  
  buffer : ARRAY[0..CONSTANTS.BufferSize] OF BYTE;
  currentBufferPos : UDINT;
  fifoHeadString : Tc2_System.T_MaxString;
  fifoHeadLength : UDINT;
  fifoHeadBytes : ARRAY[0..Tc2_System.MAX_STRING_LENGTH] OF BYTE;
  i : UINT;
END_VAR
VAR CONSTANT
  NetId : STRING := '';
  Timeout : TIME := DEFAULT_ADS_TIMEOUT;
  MaxLogsPerCycle : UINT := UDINT_TO_UINT(CONSTANTS.BufferSize / Tc2_System.MAX_STRING_LENGTH);
  MaxBufferPosition : UDINT := (SIZEOF(buffer)-Tc2_System.MAX_STRING_LENGTH);
END_VAR
// State machine
// Using if-statements instead of case for performance reasons:
// Some states execute instantly and allow thus the next state 
// to start within the same plc cycle.

// *** I D L E ***
IF state = PersistToFileState.Idle THEN
  lockFileWriteToForceRisingEdge := FALSE;
  IF _fifo.nCount > 0 AND enable THEN 
    lockFileWriteToForceRisingEdge := FALSE;
    state := PersistToFileState.OpenFile;
  END_IF
END_IF
    
// *** O P E N   F I L E ***
fileOpen(sNetId := NetId, sPathName := fileName, nMode := FOPEN_MODEAPPEND OR FOPEN_MODETEXT, 
           ePath := PATH_GENERIC, bExecute := (state = PersistToFileState.OpenFile), tTimeout := Timeout,
           hFile => fileHandle);

IF state = PersistToFileState.OpenFile THEN
  IF fileOpen.bError THEN
    state := PersistToFileState.CloseFile;
  ELSIF NOT fileOpen.bBusy THEN
    state := PersistToFileState.GetStringFromFifo; 
  END_IF
END_IF 

// *** P O P   F R O M   F I F O ***
IF state = PersistToFileState.GetStringFromFifo THEN
  IF NOT lockFileWriteToForceRisingEdge THEN
    currentBufferPos := 0;
    FOR i:=0 TO MaxLogsPerCycle DO
      IF _fifo.nCount <= 0 THEN EXIT; END_IF
      IF currentBufferPos >= MaxBufferPosition THEN EXIT; END_IF
      
      _fifo.A_RemoveHead(getValue => fifoHeadString); 
      fifoHeadBytes := MAXSTRING_TO_BYTEARR(fifoHeadString);
      fifoHeadLength := INT_TO_UDINT(LEN(fifoHeadString));
      MEMCPY(
        destAddr  :=  ADR(buffer) + SIZEOF(BYTE) * currentBufferPos,
        srcAddr   :=  ADR(fifoHeadBytes),
        n     :=  fifoHeadLength);    
      currentBufferPos := currentBufferPos + fifoHeadLength;  
    END_FOR
    state := PersistToFileState.AppendDataToFile;
  END_IF
  lockFileWriteToForceRisingEdge := FALSE;
END_IF
  
// *** W R I T E   T O   F I L E ***
fileWrite(
  sNetId := NetId, 
  hFile := fileHandle, 
  pWriteBuff := ADR(buffer),
  cbWriteLen := currentBufferPos,
  bExecute := state = PersistToFileState.AppendDataToFile, 
  tTimeout := Timeout); 

IF state = PersistToFileState.AppendDataToFile THEN
  lockFileWriteToForceRisingEdge := TRUE;   
  IF fileWrite.bError THEN
    state := PersistToFileState.CloseFile;
  ELSIF _fifo.nCount > 0 AND NOT fileWrite.bBusy THEN
    state := PersistToFileState.GetStringFromFifo; 
  ELSIF _fifo.nCount = 0 THEN
    state := PersistToFileState.CloseFile;
  END_IF
END_IF
    
// *** C L O S E   F I L E ***
fileClose(
  sNetId := NetId, hFile := fileHandle, 
  bExecute := (state = PersistToFileState.CloseFile), tTimeout := Timeout);

IF state = PersistToFileState.CloseFile THEN
  IF NOT fileClose.bBusy THEN state := PersistToFileState.Idle; END_IF
END_IF

// Close file in case of error
IF fileOpen.bError THEN state := PersistToFileState.CloseFile; END_IF
IF fileWrite.bError THEN state := PersistToFileState.CloseFile; END_IF
IF NOT _fifo.bOk AND _fifo.nCount > 0 AND state <> PersistToFileState.Idle THEN 
  state := PersistToFileState.CloseFile; 
END_IF

// Error handling
IF fileOpen.bError THEN
  Error.Active := TRUE;
  Error.Code := ErrorCodes.OpeningFileFailed;
  Error.Info := Tc2_Standard.CONCAT('Opening file failed. Error thrown by FB_FileOpen. Consult Beckhoff InfoSys. Internal Error: ', UDINT_TO_STRING(fileOpen.nErrId));
ELSIF fileWrite.bError THEN
  Error.Active := TRUE;
  Error.Code := ErrorCodes.WritingToFileFailed;
  Error.Info := Tc2_Standard.CONCAT('Writing to file failed. Error thrown by FB_FileWrite. Consult Beckhoff InfoSys. Internal Error: ', UDINT_TO_STRING(fileWrite.nErrId));
ELSIF fileClose.bError THEN
  Error.Active := TRUE;
  Error.Code := ErrorCodes.ClosingFileFailed;
  Error.Info := Tc2_Standard.CONCAT('Closing file failed. Error thrown by FB_FileClose. Consult Beckhoff InfoSys. Internal Error: ', UDINT_TO_STRING(fileClose.nErrId));
ELSIF NOT _fifo.bOk AND _fifo.nCount > 0 THEN
  Error.Active := TRUE;
  Error.Code := ErrorCodes.FifoOverflow;
  Error.Info := 'FIFO overflow. Check if plc has enough free memory.';
ELSE
  Error.Active := FALSE;
  Error.Code := ErrorCodes.None;
  Error.Info := '';
END_IF

// Set busy state
Busy := (state <> PersistToFileState.Idle OR _fifo.nCount > 0);

(* Uncomment for cyclic logging of state machine, buffer usage & errors

ADSLOGSTR(ADSLOG_MSGTYPE_LOG, 
  Tc2_Standard.CONCAT('****DynamicStringBuffer.state:', 
  Tc2_Standard.CONCAT(UINT_TO_STRING(state),
  Tc2_Standard.CONCAT(', DynamicStringBuffer.hFile:', UINT_TO_STRING(hFile)))), '');

ADSLOGSTR(ADSLOG_MSGTYPE_LOG, 
  Tc2_Standard.CONCAT('****Fifo: used ', 
  Tc2_Standard.CONCAT(UDINT_TO_STRING(Fifo.cbSize),
  Tc2_Standard.CONCAT(' of ', UDINT_TO_STRING(Fifo.cbBuffer)))), '');
  
IF Error.Active THEN
  ADSLOGSTR(ADSLOG_MSGTYPE_LOG, 
    Tc2_Standard.CONCAT('****DynamicStringBuffer.Error: ', Error.Info), 
    '');  
END_IF
*)
END_METHOD

METHOD PopHead : Tc2_System.T_MaxString
VAR_INST
  headString : Tc2_System.T_MaxString;
END_VAR
_fifo.A_RemoveHead(getValue => headString);
PopHead := headString;
END_METHOD

// Resizes the buffer for the FIFO if necessary
METHOD PRIVATE ResizeFifoBufferIfNecessary : BOOL
VAR
  requiredSize : UDINT;
  newSize : DINT;
END_VAR
requiredSize := _fifo.cbSize + (Tc2_System.MAX_STRING_LENGTH + Constants.FifoOverhead);

IF requiredSize > _fifo.cbBuffer THEN
  _dynamicMemoryBuffer.Resize(nSize := requiredSize*SIZEOF(BYTE), bPreserve:=TRUE, bReset:=TRUE);
  _fifo.pBuffer := _dynamicMemoryBuffer.pBuffer;
  _fifo.cbBuffer := requiredSize;
END_IF
END_METHOD

END_FUNCTION_BLOCK

// ---- StringBuilder/StringBuilder.TcPOU
FUNCTION_BLOCK INTERNAL StringBuilder IMPLEMENTS IStringBuilder, ILimitedStringBuilder
VAR
  {attribute 'hide'}
  _workString : Tc2_System.T_MaxString;
END_VAR

METHOD PUBLIC Append : IStringBuilder // Append text TO t current build STRING.
VAR_INPUT
  text : Tc2_System.T_MaxString; //text to append to current build string
END_VAR
_workString:= Tc2_Standard.CONCAT(_workString,text);
Append := THIS^;
END_METHOD

METHOD PUBLIC AppendIf : IStringBuilder
VAR_INPUT
  condition : BOOL;
  text : Tc2_System.T_MaxString;
END_VAR
IF condition THEN
  _workString:= Tc2_Standard.CONCAT(_workString,text);
END_IF
AppendIf := THIS^;
END_METHOD

METHOD PUBLIC InsertAtLocation : IStringBuilder
VAR_INPUT
  text : Tc2_System.T_MaxString;
  position : INT;
END_VAR
_workString := Tc2_Standard.INSERT(_workSTring,text,position);
InsertAtLocation  := THIS^;
END_METHOD

METHOD PadLeft : IStringBuilder
VAR_INPUT
  text : Tc2_System.T_MaxString; // Text to append to current build string
  length : INT; // Total length of text + padding
  c : STRING(1); // Character to be padded left of text
END_VAR
VAR
  i : INT;
  padLength : INT;
END_VAR
// Add left padding
padLength := Tc2_Standard.LEN(text) - length;
FOR i := 1 TO padLength DO
  _workString:= Tc2_Standard.CONCAT(_workString, c);
END_FOR

// Add text
_workString:= Tc2_Standard.CONCAT(_workString,text);

PadLeft := THIS^;
END_METHOD

METHOD PUBLIC Reset : ILimitedStringBuilder //Reset current build STRING TO an empty STRING.
_workString:='';
Reset := THIS^;
END_METHOD

METHOD PUBLIC ToString : Tc2_System.T_MaxString //Returns current build STRING.
ToString := _workString;
END_METHOD

END_FUNCTION_BLOCK

// ---- Utils/DateTime.TcPOU
/// Generate time data in different formats.
{attribute: 'hide_all_locals'}
FUNCTION_BLOCK DateTime
VAR
  _localSystemTime : Tc2_Utilities.FB_LocalSystemTime;
  _getSystemTime : Tc2_System.GETSYSTEMTIME;
  _timeZoneInfo : Tc2_Utilities.FB_GetTimeZoneInformation;
  _localTime : Tc2_Utilities.FB_SystemTimeToTzSpecificLocalTime;
  _localSystemTimeValid : Tc2_Standard.R_TRIG;
  _utcTime : Tc2_Utilities.FB_TzSpecificLocalTimeToFileTime;
END_VAR

// Get local system time
_localSystemTime(
  sNetID  :=  '',
  bEnable :=  TRUE,
  dwCycle :=  1,
  dwOpt :=  1,
  tTimeout:=  DEFAULT_ADS_TIMEOUT
);

// Get timezone information
_timeZoneInfo(
  sNetID := '',
  bExecute := TRUE,
  tTimeout := DEFAULT_ADS_TIMEOUT);

// Convert local time to utc time
_utcTime(
  in := THIS^.AsLocalFileTime,
  tzInfo := _timeZoneInfo.tzInfo);
  
// Finished retrieving time data
_localSystemTimeValid(CLK := _localSystemTime.bValid);

/// Returns local time as `Tc2_Utilities.T_FILETIME`.
{attribute 'monitoring':='variable'}
PROPERTY AsLocalFileTime : Tc2_Utilities.T_FILETIME
GET
AsLocalFileTime := SYSTEMTIME_TO_FILETIME(THIS^.AsLocalSystemTime);
END_GET
END_PROPERTY

/// Returns local time as `Tc2_Utilities.TIMESTRUCT`.
{attribute 'monitoring':='variable'}
PROPERTY AsLocalSystemTime : Tc2_Utilities.TIMESTRUCT
GET
AsLocalSystemTime := _localSystemTime.systemTime;
END_GET
END_PROPERTY

/// Returns local time as string.
{attribute 'monitoring':='variable'}
PROPERTY AsLocalSystemTimeString : Tc2_System.T_MAXSTRING
GET
AsLocalSystemTimeString := Tc2_Utilities.SYSTEMTIME_TO_STRING(THIS^.AsLocalSystemTime);
END_GET
END_PROPERTY

/// Returns UTC time as `Tc2_Utilities.T_FILETIME`.
{attribute 'monitoring':='variable'}
PROPERTY AsUtcFileTime : Tc2_Utilities.T_FILETIME
GET
AsUtcFileTime := _utcTime.out;
END_GET
END_PROPERTY

/// When calling `DateTime` the first time, it takes some time until all time and timezone information is available.
/// `Done` is `TRUE` for one cycle, once all the data is ready. 
{attribute 'monitoring':='call'}
PROPERTY Done : BOOL
GET
Done := _localSystemTimeValid.Q;
END_GET
END_PROPERTY

// Replaces placeholders in format string by the actual time values.
{attribute 'hide_all_locals'}
{attribute 'hide'}
METHOD PRIVATE ReplaceFormatPlaceholder : STRING
VAR_INPUT
  format : STRING;
  length : INT;
  timeType : STRING(1);
END_VAR
VAR_INST
  i : INT;
  replaceString : STRING;
  timeString : STRING;
END_VAR
VAR
  localSystemTime : Tc2_Utilities.TIMESTRUCT;
END_VAR
localSystemTime := THIS^.AsLocalSystemTime;

IF    timeType = 'Y'  THEN timeString := TO_STRING(localSystemTime.wYear); 
ELSIF timeType = 'M'  THEN timeString := TO_STRING(localSystemTime.wMonth); 
ELSIF timeType = 'D'  THEN timeString := TO_STRING(localSystemTime.wDay); 
ELSIF timeType = 'h'  THEN timeString := TO_STRING(localSystemTime.wHour); 
ELSIF timeType = 'm'  THEN timeString := TO_STRING(localSystemTime.wMinute); 
ELSIF timeType = 's'  THEN timeString := TO_STRING(localSystemTime.wSecond); 
ELSIF timeType = 'i'  THEN timeString := TO_STRING(localSystemTime.wMilliseconds); 
ELSE
  timeString:='';
END_IF

replaceString := '';

IF length > Tc2_Standard.LEN(timeString) THEN
  FOR i:=1 TO length - Tc2_Standard.LEN(timeString) DO
    replaceString := Tc2_Standard.CONCAT(replaceString, '0');
  END_FOR
  replaceString := Tc2_Standard.CONCAT(replaceString, timeString);
ELSE
  replaceString := Tc2_Standard.RIGHT(timeString, length);
END_IF

ReplaceFormatPlaceholder := Tc2_Standard.REPLACE(format, replaceString, length, Tc2_Standard.FIND(format, timeType));
END_METHOD

/// Returns a formatted string containing the actual time information 
/// - `Y` : year
/// - `M` : month
/// - `D` : day
/// - `h` : hour 
/// - `m` : minute
/// - `s` : second
/// - `i` : millisecond
/// 
/// Example:    
/// _YYMMDD-hh:mm:ss:iii_   
/// => _20210812-12:30:22:123_
{attribute 'hide_all_locals'}
METHOD ToFormatString : Tc2_System.T_MaxString
VAR_INPUT
  /// Format the timestamp should have.
  format : STRING;
END_VAR
VAR_INST
  inputString : STRING;
  c : STRING(1);
  formattedString : Tc2_System.T_MaxString;
END_VAR
VAR
  year : INT := 0;
  month : INT := 0;
  day : INT := 0;
  hour : INT := 0;
  minute : INT := 0;
  second : INT := 0;
  millisecond : INT := 0;
END_VAR
VAR CONSTANT
  ValidFormat : STRING := 'YMDhms';
END_VAR
// Parses "format" and returns a adequatly formatted string containing the time information
inputString := format;

WHILE Tc2_Standard.LEN(inputString) > 0 DO
  c := Tc2_Standard.LEFT(inputString, 1);
  
  IF    c = 'Y' THEN year := year + 1;
  ELSIF c = 'M' THEN month := month + 1;
  ELSIF c = 'D' THEN day := day + 1;
  ELSIF c = 'h' THEN hour := hour + 1;
  ELSIF c = 'm' THEN minute := minute + 1;
  ELSIF c = 's' THEN second := second + 1;
  ELSIF c = 'i' THEN millisecond := millisecond + 1;
  END_IF
  
  inputString := Tc2_Standard.DELETE(inputString, 1, 1);
END_WHILE

formattedString := ReplaceFormatPlaceholder(format, year, 'Y');
formattedString := ReplaceFormatPlaceholder(formattedString, month, 'M');
formattedString := ReplaceFormatPlaceholder(formattedString, day, 'D');
formattedString := ReplaceFormatPlaceholder(formattedString, hour, 'h');
formattedString := ReplaceFormatPlaceholder(formattedString, minute, 'm');
formattedString := ReplaceFormatPlaceholder(formattedString, second, 's');
formattedString := ReplaceFormatPlaceholder(formattedString, millisecond, 'i');

ToFormatString := formattedString;
END_METHOD

END_FUNCTION_BLOCK

// ---- Utils/DeleteOldFiles.TcPOU
{attribute 'hide_all_locals'}
FUNCTION_BLOCK INTERNAL DeleteOldFiles
VAR_INPUT
  StartScan : BOOL; // Rising edge starts scan for out-of-date log files and deletes them.
  ExpirationInDays : UINT; // Files will be deleted if older than n days
  FilePath : Tc2_System.T_MaxString; // Path to files to be deleted
  FileName : Tc2_System.T_MaxString; // Only files which match this filename will be deleted
  CurrentUtcTime : Tc2_Utilities.T_FILETIME; // Current time  as UTC
END_VAR
VAR_OUTPUT
  Error : Error; // Error information
END_VAR
VAR CONSTANT
  OneDayInSeconds : LREAL := 24*3600.0;
  MaxNumberOfFiles : UDINT := 100;
END_VAR
VAR
  _state : DeleteFilesState := DeleteFilesState.Idle;
  
  _enumFindFileList : Tc2_Utilities.FB_EnumFindFileList;
  _enumBusy : Tc2_Standard.F_TRIG;
  _fileDelete : Tc2_System.FB_FileDelete;
  _fileDeleteBusy : Tc2_Standard.F_TRIG;
  _listOfFiles : ARRAY[1..100] OF Tc2_Utilities.ST_FindFileEntry;
  _deleteFileIndex : UDINT;
  _fileNameToDelete : Tc2_System.T_MaxString;
  _commandType : Tc2_Utilities.E_EnumCmdType;
  _fileDeleted : BOOL;
  _startFileDelete: BOOL;
END_VAR

// State machine to delete all due files.
// It first enumerates all files in the specified directory
// and then deletes all files that have overpassed the specified due date
_startFileDelete := FALSE;

CASE _state OF
  DeleteFilesState.Idle:
    IF StartScan THEN
      _commandType:= eEnumCmd_First;
      _deleteFileIndex := 1;
      _state := DeleteFilesState.SearchNextFile;
    END_IF
    
  DeleteFilesState.SearchNextFile:
    IF _enumBusy.Q THEN
      _state := DeleteFilesState.WaitUntilExecutionDone;
    END_IF
    
  DeleteFilesState.WaitUntilExecutionDone:
    IF NOT _enumFindFileList.bError THEN
      IF NOT _enumFindFileList.bEOE THEN
        IF _enumFindFileList.nFindFiles < MaxNumberOfFiles THEN
          _state := DeleteFilesState.SearchNextFile;
        ELSE
          _commandType := eEnumCmd_Abort;
          _state := DeleteFilesState.ProcessFoundFiles;
        END_IF
      ELSE
        _state := DeleteFilesState.ProcessFoundFiles;
      END_IF
    ELSE
      _state := DeleteFilesState.Idle;
    END_IF
    
  DeleteFilesState.ProcessFoundFiles:
    IF _deleteFileIndex > _enumFindFileList.nFindFiles THEN
      _state := DeleteFilesState.Idle;
    ELSE
      _state := DeleteFilesState.CheckIfFileIsDirectory;
    END_IF
    
  DeleteFilesState.CheckIfFileIsDirectory:
    IF NOT _listOfFiles[_deleteFileIndex].fileAttributes.bDirectory THEN
      _state := DeleteFilesState.CheckFileTime;
    ELSE
      _deleteFileIndex := _deleteFileIndex + 1;
      _state := DeleteFilesState.ProcessFoundFiles;
    END_IF
    
  DeleteFilesState.CheckFileTime:   
    IF GetFileAgeInSeconds(CurrentUtcTime, _listOfFiles[_deleteFileIndex]) > (ExpirationInDays * OneDayInSeconds) THEN
      _state := DeleteFilesState.DeleteFile;
    ELSE
      _deleteFileIndex := _deleteFileIndex + 1;
      _state := DeleteFilesState.ProcessFoundFiles;
    END_IF
  
  DeleteFilesState.DeleteFile:
    _fileNameToDelete := Tc2_Standard.CONCAT(FilePath, _listOfFiles[_deleteFileIndex].sFileName);
    _startFileDelete := TRUE;
    
    IF _fileDeleteBusy.Q THEN
      _deleteFileIndex := _deleteFileIndex + 1;
      _fileDeleted := TRUE;
      _state := DeleteFilesState.FileDeleted;
    END_IF
    IF _fileDelete.bError THEN
      _state := DeleteFilesState.Idle;
    END_IF
    
  DeleteFilesState.FileDeleted:   
    // This state is needed to generate a rising edge for FB_FileDelete
    IF NOT _fileDeleted THEN
      _state := DeleteFilesState.ProcessFoundFiles;
    END_IF
    _fileDeleted := FALSE;

END_CASE

// Function blocks used in state machine

// Search files in given directory
_enumFindFileList(sNetId := '',
       eCmd := _commandType,
       sPathName := Tc2_Standard.CONCAT(FilePath, Tc2_Standard.CONCAT('*', FileName)),
       bExecute := (_state = DeleteFilesState.SearchNextFile) OR (_commandType = eEnumCmd_Abort AND _state <> DeleteFilesState.Idle),
       pFindList := ADR(_listOfFiles),
       cbFindList := SIZEOF(_listOfFiles),
       tTimeout := T#10S);
       
_enumBusy(CLK:=_enumFindFileList.bBusy);

// Delete files
_fileDelete(sNetId := '',
             sPathName := _fileNameToDelete,
             bExecute := _startFileDelete,
             tTimeout := T#10S);

_fileDeleteBusy(CLK := _fileDelete.bBusy);

// Error handling
Error.Active := FALSE;
Error.Code := ErrorCodes.None;
Error.Info := '';

IF _enumFindFileList.bError THEN
  Error.Active := TRUE;
  Error.Code := ErrorCodes.EnumeratingFilesInSpecifiedDirectoryFailed;
  Error.Info := Tc2_Standard.CONCAT('Enumerating files in specified directory failed. Error thrown by FB_EnumFindFileList. Consult Beckhoff InfoSys. Internal Error: ', UDINT_TO_STRING(_enumFindFileList.nErrId));
END_IF
      
IF _fileDelete.bError THEN
  Error.Active := TRUE;
  Error.Code := ErrorCodes.DeletingFileFailed;
  Error.Info := Tc2_Standard.CONCAT('Deleting expired log file in specified directory failed. Error thrown by FB_FileDelete. Consult Beckhoff InfoSys. Internal Error: ', UDINT_TO_STRING(_fileDelete.nErrId));
END_IF

END_FUNCTION_BLOCK

// ---- Utils/GetFileAgeInSeconds.TcPOU
{attribute 'hide'}
FUNCTION INTERNAL GetFileAgeInSeconds : DINT
VAR_INPUT
  currentUtcTime : Tc2_Utilities.T_FILETIME;
  findFileEntry : Tc2_Utilities.ST_FindFileEntry;
END_VAR
VAR
  _timeLastWriteAccess : Tc2_Utilities.T_ULARGE_INTEGER;
  _fileTimeAsULINT : Tc2_Utilities.T_ULARGE_INTEGER;
  _fileTimeDifference : Tc2_Utilities.T_ULARGE_INTEGER;
END_VAR
VAR CONSTANT
  OneSecondInOneHundredNanoSecondsIntervals : LREAL := 1000*1000*10;
END_VAR

// Local file time
_fileTimeAsULINT.dwLowPart := currentUtcTime.dwLowDateTime;
_fileTimeAsULINT.dwHighPart := currentUtcTime.dwHighDateTime;

// Write access is UTC
_timeLastWriteAccess.dwLowPart := findFileEntry.lastWriteTime.dwLowDateTime;
_timeLastWriteAccess.dwHighPart := findFileEntry.lastWriteTime.dwHighDateTime;
_fileTimeDifference := UInt64Sub64(_fileTimeAsULINT, _timeLastWriteAccess);

GetFileAgeInSeconds := LREAL_TO_DINT(UINT64_TO_LREAL(_fileTimeDifference)/(OneSecondInOneHundredNanoSecondsIntervals));

END_FUNCTION

// ---- Logger/TcLogTrig.TcPOU
/// This function block can be used to log on rising or falling edges.
/// For each signal that should be watched, a separate instance of `TcLogTrig` 
/// must be created.
FUNCTION_BLOCK TcLogTrig EXTENDS TcLog

/// Logs data on falling edge of `CLK`.
{attribute 'hide_all_locals'}
METHOD OnFallingEdge : REFERENCE TO TcLog
VAR_INPUT
  /// Falling edge triggers logging the data.
  CLK : BOOL; 
END_VAR
VAR_INST
    fTrig : Tc2_Standard.F_TRIG;
END_VAR
fTrig(CLK:=CLK);

SUPER^.OnCondition(fTrig.Q);

OnFallingEdge REF= THIS^;
END_METHOD

/// Logs data on rising edge of `CLK`.
{attribute 'hide_all_locals'}
METHOD OnRisingEdge : REFERENCE TO TcLog
VAR_INPUT
  /// Rising edge logs data.
  CLK : BOOL; 
END_VAR
VAR_INST
    rTrig : Tc2_Standard.R_TRIG;
END_VAR
rTrig(CLK:=CLK);

SUPER^.OnCondition(rTrig.Q);

OnRisingEdge REF= THIS^;
END_METHOD

END_FUNCTION_BLOCK

// ---- Logger/_Tests/TestWrapper_NET.TcPOU
FUNCTION_BLOCK TestWrapper_NET
VAR
  _coreLogger : TcLogCore(BufferSize:=50 * 50 * (Tc2_System.MAX_STRING_LENGTH + Constants.FifoOverhead));
  _coreLoggerFirstCycle : TcLogCore(BufferSize:=50 * 50 * (Tc2_System.MAX_STRING_LENGTH + Constants.FifoOverhead));
  _coreLoggerFirstCycleValidTimestampOnly : TcLogCore(BufferSize:=50 * 50 * (Tc2_System.MAX_STRING_LENGTH + Constants.FifoOverhead));
  _loggerFirstCycle : TcLog;
  _loggerFirstCycleValidTimestampOnly : TcLog;
  _logger : TcLog;
  _flushCache : BOOL;
 
  // Test drivers
  _getDateTime : DateTime;
  _setLocalSystemTime : NT_SetLocalTime;
  _cycles : INT;
  _i : INT;
  _persistenceTimeStaysWithinBounds : F_TRIG;
  _isFirstCycle: BOOL := TRUE;
  
  // Exchanged variables with .NET tests
  FilePath : STRING;
  FileName : STRING;
  Delimiter : STRING(1);
  NewLocalSystemTimeToBeSet : STRING;
  TriggerNewLocalSystemTime : BOOL;
  LocalTimeAsString : STRING;
  
  Persist_simple_error_message_run : BOOL;
  Persist_simple_error_message_data : STRING;
  
  Persist_long_error_message_run : BOOL;
  Persist_long_error_message_data : T_MaxString;
  
  Linebreak_is_included_when_log_message_has_maximum_length_run : BOOL;
  Linebreak_is_included_when_log_message_has_maximum_length_data : T_MaxString;
  
  Do_not_persist_logs_below_log_level_run : BOOL;
  
  Log_message_contains_instance_path_run : BOOL;
  
  Log_message_uses_correct_delimiter_run : BOOL;
  Log_message_uses_correct_delimiter_data : STRING;
  
  Log_message_contains_custom_formatted_timestamp_run : BOOL;
  
  Delete_logs_if_expired_run : BOOL;
  
  New_logfile_is_created_if_rolling_interval_rolls_run : BOOL;
  
  Same_log_file_is_used_until_rolling_interval_rolls : BOOL;
  
  Log_in_consecutive_cycles : BOOL;
  Number_of_log_cycles : DINT;
  
  Log_multiple_logs_in_one_cycle : BOOL;
  Number_of_logs_per_cycle : DINT;
  
  Log_multiple_logs_in_multiple_cycles : BOOL;
  Number_of_cycles : DINT;
  CycleCount : DINT := 1;
  
  Persistance_time_stays_within_bounds : BOOL;
  Duration_in_cylces : DINT := 1;
  
END_VAR

// ****** U N I T   T E S T S ******

// Set up TcLog
_coreLogger
  .IncludeInstancePath()
  .MinimumLevel(LogLevels.Warning)
  .SetDelimiter(Delimiter)
  .SetRollingInterval(RollingIntervals.Hourly)
  .DeleteLogFilesAfterDays(1)
  .TimestampFormat('_YYMMDD-hh-mm-ss_')
  .WriteToAds()
  .WriteToFile(FilePath, FileName)
  .RunLogger();
//_logger.SetLogger(_coreLogger);

IF _flushCache THEN _coreLogger.FlushCache(); END_IF
  
// Test drivers
_getDateTime();
LocalTimeAsString := _getDateTime.AsLocalSystemTimeString;

_setLocalSystemTime(
  NETID   := '',
  TIMESTR := STRING_TO_SYSTEMTIME(NewLocalSystemTimeToBeSet),
  START   := TriggerNewLocalSystemTime,
  TMOUT := T#2S
  );

// Execute tests
IF Persist_simple_error_message_run THEN
  Persist_simple_error_message_run := FALSE;
  _logger
    .Error(Persist_simple_error_message_data);
END_IF

IF Persist_long_error_message_run THEN
  Persist_long_error_message_run := FALSE;
  _logger
    .ToCustomFormat(Persist_long_error_message_data);
END_IF

IF Linebreak_is_included_when_log_message_has_maximum_length_run THEN
  Linebreak_is_included_when_log_message_has_maximum_length_run := FALSE;
  _logger
    .ToCustomFormat(Linebreak_is_included_when_log_message_has_maximum_length_data);
  _logger
    .ToCustomFormat(Linebreak_is_included_when_log_message_has_maximum_length_data);
END_IF


IF Do_not_persist_logs_below_log_level_run THEN
  Do_not_persist_logs_below_log_level_run := FALSE;
  _logger
    .Information('Nothing');
END_IF

IF Log_message_contains_instance_path_run THEN
  Log_message_contains_instance_path_run := FALSE;
  _logger
    .Error('Nothing');
END_IF

IF Log_message_uses_correct_delimiter_run THEN
  Log_message_uses_correct_delimiter_run := FALSE;
  _logger
    .Error(Log_message_uses_correct_delimiter_data);
END_IF

IF Log_message_contains_custom_formatted_timestamp_run THEN
  Log_message_contains_custom_formatted_timestamp_run := FALSE;
  _logger
    .Error('Test message');
END_IF

IF Delete_logs_if_expired_run THEN
  Delete_logs_if_expired_run := FALSE;
  _logger
    .Error('Test message');
END_IF

IF New_logfile_is_created_if_rolling_interval_rolls_run THEN
  New_logfile_is_created_if_rolling_interval_rolls_run := FALSE;
  _logger
    .Error('Test message');
END_IF

IF Same_log_file_is_used_until_rolling_interval_rolls THEN
  Same_log_file_is_used_until_rolling_interval_rolls := FALSE;
  _logger
    .Error('Test message');
END_IF

IF Log_in_consecutive_cycles THEN
  _logger
    .Error(Tc2_Standard.CONCAT('Logging cycle ', INT_TO_STRING(_cycles)));
  _cycles := _cycles + 1;
  IF _cycles >= Number_of_log_cycles THEN
    _cycles := 0;
    Log_in_consecutive_cycles := FALSE;
  END_IF
END_IF

IF Log_multiple_logs_in_one_cycle THEN
  FOR _i:= 1 TO DINT_TO_INT(Number_of_logs_per_cycle) DO
    _logger.
      Error(Tc2_Standard.CONCAT('Logging multiple times per cycle. Current step: ', INT_TO_STRING(_i))); 
  END_FOR
  Log_multiple_logs_in_one_cycle := FALSE;
END_IF

IF Log_multiple_logs_in_multiple_cycles THEN
  IF CycleCount <= Number_of_cycles THEN  
    FOR _i:= 1 TO DINT_TO_INT(Number_of_logs_per_cycle) DO
      _logger
        .AppendString('Logging multiple times per cycle. Cycle: ')
        .AppendString(DINT_TO_STRING(CycleCount))
        .AppendString(' / Step: ')
        .AppendString(INT_TO_STRING(_i))
        .Error('');
    END_FOR
    CycleCount := CycleCount + 1;
  ELSE
    CycleCount := 1;
    Log_multiple_logs_in_multiple_cycles := FALSE;
  END_IF
END_IF 

_persistenceTimeStaysWithinBounds(CLK := (Persistance_time_stays_within_bounds AND _coreLogger.Busy));
IF _persistenceTimeStaysWithinBounds.Q THEN
  CycleCount := 1;
  Persistance_time_stays_within_bounds := FALSE;
END_IF
IF Persistance_time_stays_within_bounds THEN
  Duration_in_cylces := Duration_in_cylces + 1;
  IF CycleCount <= Number_of_cycles THEN  
    FOR _i:= 1 TO DINT_TO_INT(Number_of_logs_per_cycle) DO
      _logger
        .AppendString('Logging multiple times per cycle. Cycle: ')
        .AppendString(DINT_TO_STRING(CycleCount))
        .AppendString(' / Step: ')
        .AppendString(INT_TO_STRING(_i))
        .Error('');
    END_FOR
    CycleCount := CycleCount + 1;
  END_IF
END_IF

// Check first cpu cycle
_coreLoggerFirstCycle
  .IncludeInstancePath()
  .MinimumLevel(LogLevels.Warning)
  .SetDelimiter(Delimiter)
  .SetRollingInterval(RollingIntervals.Hourly)
  .DeleteLogFilesAfterDays(1)
  .TimestampFormat('_YYYYMMDD-hh-mm-ss_')
  .WriteToAds()
  .WriteToFile('C:\UnitTestFirstCycle\', 'firstCycle.txt')
  .RunLogger();
_loggerFirstCycle.SetLogger(_coreLoggerFirstCycle);

_coreLoggerFirstCycleValidTimestampOnly
  .IncludeInstancePath()
  .MinimumLevel(LogLevels.Warning)
  .SetDelimiter(Delimiter)
  .SetRollingInterval(RollingIntervals.Hourly)
  .DeleteLogFilesAfterDays(1)
  .TimestampFormat('_YYYYMMDD-hh-mm-ss_')
  .WriteToAds()
  .WriteToFile('C:\UnitTestFirstCycle\', 'firstCycleValidTimestampOnly.txt')
  .ValidTimestampsOnly()
  .RunLogger();
_loggerFirstCycleValidTimestampOnly.SetLogger(_coreLoggerFirstCycleValidTimestampOnly);

IF _isFirstCycle THEN
  _loggerFirstCycle.Error('Log in first cycle');
  _loggerFirstCycleValidTimestampOnly.Error('Log in first cycle');
  _isFirstCycle := FALSE;
END_IF

END_FUNCTION_BLOCK

// ---- Utils/_Tests/ConvertAnyToString_TEST.TcPOU
FUNCTION_BLOCK ConvertAnyToString_TEST EXTENDS TcUnit.FB_TestSuite

ConvertAnyByteToString();
ConvertAnyDateAndTimeToString();
ConvertAnyDateToString();
ConvertAnyDINTToString();
ConvertAnyDTToString();
ConvertAnyINTToString();
ConvertAnyLINTToString();
//ConvertAnyLRealToString();
ConvertAnyLWordToString();
ConvertAnyRealToString();
ConvertAnySINTToString();
ConvertAnyStringToString();
ConvertAnyTimeToString();
ConvertAnyTODToString();
ConvertAnyUDINTToString();
ConvertAnyUINTToString();
ConvertAnyULINTToString();
ConvertAnyUSINTToString();
ConvertAnyWordToString();
ConvertAnyWStringToString();

METHOD ConvertAnyByteToString : BOOL
VAR
  inputs : ARRAY[1..4] OF BYTE := [0, 1, 128, 255];
  expectedValues : ARRAY[1..4] OF STRING := ['0', '1', '128', '255'];
  results : ARRAY[1..4] OF STRING;
  i: INT;
END_VAR
TEST('ConvertAnyByteToString');
 
FOR i := 1 TO 4 DO
  results[i] := AnyToString(inputs[i]);
  AssertEquals(Expected := expectedValues[i],
             Actual := results[i],
             Message := FormatResult(expectedValues[i], results[i])); 
END_FOR
 
TEST_FINISHED();
END_METHOD

METHOD ConvertAnyDateAndTimeToString : BOOL
VAR
  input : DATE_AND_TIME := DT#1970-01-01-00:00;
  result : STRING;
  expected : STRING := 'DT#1970-01-01-00:00:00';
END_VAR
TEST('ConvertAnyDateAndTimeToString');
 
result := AnyToString(input);
 
AssertEquals(Expected := expected,
             Actual := result,
             Message := FormatResult(expected, result));
 
TEST_FINISHED();
END_METHOD

METHOD ConvertAnyDateToString : BOOL
VAR
  input : DATE := D#1970-01-01;
  result : STRING;
  expected : STRING := 'D#1970-01-01';
END_VAR
TEST('ConvertAnyDateToString');
 
result := AnyToString(input);
 
AssertEquals(Expected := expected,
             Actual := result,
             Message := FormatResult(expected, result));
 
TEST_FINISHED();
END_METHOD

METHOD ConvertAnyDINTToString : BOOL
VAR
  inputs : ARRAY[1..7] OF DINT := [-2147483648, -1073741824, -1, 0, 1, 1073741824, 2147483647];
  expectedValues : ARRAY[1..7] OF STRING := ['-2147483648', '-1073741824', '-1', '0', '1', '1073741824', '2147483647'];
  results : ARRAY[1..7] OF STRING;
  i: INT;
END_VAR
TEST('ConvertAnyDINTToString');
 
FOR i := 1 TO 7 DO
  results[i] := AnyToString(inputs[i]);
  AssertEquals(Expected := expectedValues[i],
             Actual := results[i],
             Message := FormatResult(expectedValues[i], results[i])); 
END_FOR

TEST_FINISHED();
END_METHOD

METHOD ConvertAnyDTToString : BOOL
VAR
  input : DT := DT#1970-01-01-00:00;
  result : STRING;
  expected : STRING := 'DT#1970-01-01-00:00:00';
END_VAR
TEST('ConvertAnyDTToString');
 
result := AnyToString(input);
 
AssertEquals(Expected := expected,
             Actual := result,
             Message := FormatResult(expected, result));
 
TEST_FINISHED();
END_METHOD

METHOD ConvertAnyDWordToString : BOOL
VAR
  inputs : ARRAY[1..4] OF DWORD := [0, 1, 2147483647, 4294967295];
  expectedValues : ARRAY[1..4] OF STRING := ['0', '1', '2147483647', '4294967295'];
  results : ARRAY[1..4] OF STRING;
  i: INT;
END_VAR
TEST('ConvertAnyDWordToString');
 
FOR i := 1 TO 4 DO
  results[i] := AnyToString(inputs[i]);
  AssertEquals(Expected := expectedValues[i],
             Actual := results[i],
             Message := FormatResult(expectedValues[i], results[i])); 
END_FOR
 
TEST_FINISHED();
END_METHOD

METHOD ConvertAnyINTToString : BOOL
VAR
  inputs : ARRAY[1..7] OF INT := [-32768, -18000, -1, 0, 1, 18000, 32767];
  expectedValues : ARRAY[1..7] OF STRING := ['-32768', '-18000', '-1', '0', '1', '18000', '32767'];
  results : ARRAY[1..7] OF STRING;
  i: INT;
END_VAR
TEST('ConvertAnyINTToString');

FOR i := 1 TO 7 DO
  results[i] := AnyToString(inputs[i]);
  AssertEquals(Expected := expectedValues[i],
             Actual := results[i],
             Message := FormatResult(expectedValues[i], results[i])); 
END_FOR
      
TEST_FINISHED();
END_METHOD

METHOD ConvertAnyLINTToString : BOOL
VAR
  inputs : ARRAY[1..7] OF LINT := [-2147483648, -18000, -1, 0, 1, 18000, 2147483648];
  expectedValues : ARRAY[1..7] OF STRING := ['-2147483648', '-18000', '-1', '0', '1', '18000', '2147483648'];
  results : ARRAY[1..7] OF STRING;
  i: INT;
END_VAR
TEST('ConvertAnyLINTToString');
 
FOR i := 1 TO 7 DO
  results[i] := AnyToString(inputs[i]);
  AssertEquals(Expected := expectedValues[i],
             Actual := results[i],
             Message := FormatResult(expectedValues[i], results[i])); 
END_FOR
 
TEST_FINISHED();
END_METHOD

METHOD ConvertAnyLRealToString : BOOL
VAR
  inputs : ARRAY[1..5] OF LREAL := [-1.7976931348623157E+308, -4.94065645841247E-324, 0, 4.94065645841247E-324, 1.7976931348623157E+308];
  expectedValues : ARRAY[1..5] OF STRING := ['-1.7976931348623157E308', '-4.94065645841247E324', '0.0', '4.94065645841247E324', '1.7976931348623157E308'];
  results : ARRAY[1..5] OF STRING;
  i: INT;
END_VAR
TEST('ConvertAnyRealToString');
 
FOR i := 1 TO 5 DO
  results[i] := AnyToString(inputs[i]);
  AssertEquals(Expected := expectedValues[i],
             Actual := results[i],
             Message := FormatResult(expectedValues[i], results[i])); 
END_FOR
 
TEST_FINISHED();
END_METHOD

METHOD ConvertAnyLWordToString : BOOL
VAR
  inputs : ARRAY[1..4] OF LWORD := [0, 1, 2147483647, 4294967295];
  expectedValues : ARRAY[1..4] OF STRING := ['0', '1', '2147483647', '4294967295'];
  results : ARRAY[1..4] OF STRING;
  i: INT;
END_VAR
TEST('ConvertAnyLWordToString');
 
FOR i := 1 TO 4 DO
  results[i] := AnyToString(inputs[i]);
  AssertEquals(Expected := expectedValues[i],
             Actual := results[i],
             Message := FormatResult(expectedValues[i], results[i])); 
END_FOR

TEST_FINISHED();
END_METHOD

METHOD ConvertAnyRealToString : BOOL
VAR
  inputs : ARRAY[1..5] OF REAL := [-3.402823E+38, -1.0, 0, 1.0, 3.402823E+38];
  expectedValues : ARRAY[1..5] OF STRING := ['-3.402823E38', '-1.0', '0.0', '1.0', '3.402823E38'];
  results : ARRAY[1..5] OF STRING;
  i: INT;
END_VAR
TEST('ConvertAnyRealToString');
 
FOR i := 1 TO 5 DO
  results[i] := AnyToString(inputs[i]);
  AssertEquals(Expected := expectedValues[i],
             Actual := results[i],
             Message := FormatResult(expectedValues[i], results[i])); 
END_FOR
 
TEST_FINISHED();
END_METHOD

METHOD ConvertAnySINTToString : BOOL
VAR
  inputs : ARRAY[1..5] OF SINT := [-128, -1, 0, 1, 127];
  expectedValues : ARRAY[1..5] OF STRING := ['-128', '-1', '0', '1', '127'];
  results : ARRAY[1..5] OF STRING;
  i: INT;
END_VAR
TEST('ConvertAnySINTToString');
 
FOR i := 1 TO 5 DO
  results[i] := AnyToString(inputs[i]);
  AssertEquals(Expected := expectedValues[i],
             Actual := results[i],
             Message := FormatResult(expectedValues[i], results[i])); 
END_FOR
 
TEST_FINISHED();
END_METHOD

METHOD ConvertAnyStringToString : BOOL
VAR
  input : STRING := 'Hallo';
  result : STRING;
  expected : STRING := 'Hallo';
END_VAR
TEST('ConvertAnyStringToString');
 
result := AnyToString(input);
 
AssertEquals(Expected := expected,
             Actual := result,
             Message := FormatResult(expected, result));
 
TEST_FINISHED();
END_METHOD

METHOD ConvertAnyTimeToString : BOOL
VAR
  input : TIME := T#49D17H2M47S295MS;
  result : STRING;
  expected : STRING := 'T#49d17h2m47s295ms';
END_VAR
TEST('ConvertAnyTimeToString');
 
result := AnyToString(input);
 
AssertEquals(Expected := expected,
             Actual := result,
             Message := FormatResult(expected, result));
 
TEST_FINISHED();
END_METHOD

METHOD ConvertAnyTODToString : BOOL
VAR
  input : TOD := TOD#11:02:47.295;
  result : STRING;
  expected : STRING := 'TOD#11:02:47.295';
END_VAR
TEST('ConvertAnyTODToString');
 
result := AnyToString(input);
 
AssertEquals(Expected := expected,
             Actual := result,
             Message := FormatResult(expected, result));
 
TEST_FINISHED();
END_METHOD

METHOD ConvertAnyUDINTToString : BOOL
VAR
  inputs : ARRAY[1..3] OF UDINT := [0, 1, 4294967295];
  expectedValues : ARRAY[1..3] OF STRING := ['0', '1', '4294967295'];
  results : ARRAY[1..3] OF STRING;
  i: INT;
END_VAR
TEST('ConvertAnyUDINTToString');

FOR i := 1 TO 3 DO
  results[i] := AnyToString(inputs[i]);
  AssertEquals(Expected := expectedValues[i],
             Actual := results[i],
             Message := FormatResult(expectedValues[i], results[i])); 
END_FOR
 
TEST_FINISHED();
END_METHOD

METHOD ConvertAnyUINTToString : BOOL
VAR
  inputs : ARRAY[1..3] OF UINT := [0, 1, 65535];
  expectedValues : ARRAY[1..3] OF STRING := ['0', '1', '65535'];
  results : ARRAY[1..3] OF STRING;
  i: INT;
END_VAR
TEST('ConvertAnyUINTToString');
 
FOR i := 1 TO 3 DO
  results[i] := AnyToString(inputs[i]);
  AssertEquals(Expected := expectedValues[i],
             Actual := results[i],
             Message := FormatResult(expectedValues[i], results[i])); 
END_FOR
 
TEST_FINISHED();
END_METHOD

METHOD ConvertAnyULINTToString : BOOL
VAR
  inputs : ARRAY[1..3] OF ULINT := [0, 1, 4294967295];
  expectedValues : ARRAY[1..3] OF STRING := ['0', '1', '4294967295'];
  results : ARRAY[1..3] OF STRING;
  i: INT;
END_VAR
TEST('ConvertAnyULINTToString');
 
FOR i := 1 TO 3 DO
  results[i] := AnyToString(inputs[i]);
  AssertEquals(Expected := expectedValues[i],
             Actual := results[i],
             Message := FormatResult(expectedValues[i], results[i])); 
END_FOR
 
TEST_FINISHED();
END_METHOD

METHOD ConvertAnyUSINTToString : BOOL
VAR
  inputs : ARRAY[1..3] OF USINT := [0, 1, 255];
  expectedValues : ARRAY[1..3] OF STRING := ['0', '1', '255'];
  results : ARRAY[1..3] OF STRING;
  i: INT;
END_VAR
TEST('ConvertAnyUSINTToString');
 
FOR i := 1 TO 3 DO
  results[i] := AnyToString(inputs[i]);
  AssertEquals(Expected := expectedValues[i],
             Actual := results[i],
             Message := FormatResult(expectedValues[i], results[i])); 
END_FOR
 
TEST_FINISHED();
END_METHOD

METHOD ConvertAnyWordToString : BOOL
VAR
  inputs : ARRAY[1..3] OF WORD := [0, 1, 65535];
  expectedValues : ARRAY[1..3] OF STRING := ['0', '1', '65535'];
  results : ARRAY[1..3] OF STRING;
  i: INT;
END_VAR
TEST('ConvertAnyWordToString');
 
FOR i := 1 TO 3 DO
  results[i] := AnyToString(inputs[i]);
  AssertEquals(Expected := expectedValues[i],
             Actual := results[i],
             Message := FormatResult(expectedValues[i], results[i])); 
END_FOR
 
TEST_FINISHED();
END_METHOD

METHOD ConvertAnyWStringToString : BOOL
VAR
  input : WSTRING := "Hallo";
  result : STRING;
  expected : STRING := 'Hallo';
END_VAR
TEST('ConvertAnyWStringToString');
 
result := AnyToString(input);
 
AssertEquals(Expected := expected,
             Actual := result,
             Message := FormatResult(expected, result));
 
TEST_FINISHED();
END_METHOD

METHOD PRIVATE FormatResult : STRING
VAR_INPUT
  Expected : STRING;
  Result : STRING;
END_VAR
FormatResult := Tc2_Standard.CONCAT('Conversion failed. Expected: ', Tc2_Standard.CONCAT(Expected, Tc2_Standard.CONCAT(' - Result: ', Result)));
END_METHOD

END_FUNCTION_BLOCK

// ---- Utils/_Tests/DateTime_TEST.TcPOU
FUNCTION_BLOCK DateTime_TEST EXTENDS TcUnit.FB_TestSuite

CheckStringFormat();

METHOD CheckStringFormat
VAR_INST
  sut : DateTime;
  expected : STRING;
  result : STRING;
END_VAR
VAR
  localSystemTime : Tc2_Utilities.TIMESTRUCT;
END_VAR
sut();

TEST('CheckStringFormat');

localSystemTime := sut.AsLocalSystemTime;

expected := Tc2_Standard.CONCAT('-', TO_STRING(localSystemTime.wYear));
IF localSystemTime.wMonth < 10 THEN expected := Tc2_Standard.CONCAT(expected, '0'); END_IF
expected := Tc2_Standard.CONCAT(expected, TO_STRING(localSystemTime.wMonth));
IF localSystemTime.wDay < 10 THEN expected := Tc2_Standard.CONCAT(expected, '0'); END_IF
expected := Tc2_Standard.CONCAT(expected, TO_STRING(localSystemTime.wDay));
expected := Tc2_Standard.CONCAT(expected, '-');
IF localSystemTime.wHour < 10 THEN expected := Tc2_Standard.CONCAT(expected, '0'); END_IF
expected := Tc2_Standard.CONCAT(expected, TO_STRING(localSystemTime.wHour));
expected := Tc2_Standard.CONCAT(expected, ':');
IF localSystemTime.wMinute < 10 THEN expected := Tc2_Standard.CONCAT(expected, '0'); END_IF
expected := Tc2_Standard.CONCAT(expected, TO_STRING(localSystemTime.wMinute));
expected := Tc2_Standard.CONCAT(expected, ':');
IF localSystemTime.wSecond < 10 THEN expected := Tc2_Standard.CONCAT(expected, '0'); END_IF
expected := Tc2_Standard.CONCAT(expected, TO_STRING(localSystemTime.wSecond));
expected := Tc2_Standard.CONCAT(expected, '-');

result := sut.ToFormatString('-YYYYMMDD-hh:mm:ss-');
  
IF sut.Done THEN
  AssertEquals(
    Expected  :=  expected,
    Actual    :=  result,
    Message   :=  'Time formatting failed.'
  );

  TEST_FINISHED();
END_IF
END_METHOD

END_FUNCTION_BLOCK

// ---- Utils/_Tests/DynamicStringBuffer_TEST.TcPOU
FUNCTION_BLOCK DynamicStringBuffer_TEST EXTENDS FB_TestSuite

LogsManyMessagesForManyCycles();

METHOD LogsManyMessagesForManyCycles
VAR
  result : STRING := '';
  expected : STRING := '';
  i : UDINT;
END_VAR
VAR CONSTANT
  Cycles : UDINT := 50;
  Messages : UDINT := 50;
END_VAR
VAR_INST
  cycleCount : UDINT := 0;
  logsManyMessagesForManyCyclesLogger : TcLogCore(BufferSize:=50 * 50 * 280); // Cycles * Messages * (max string length + fifo overhead (estimated))
  logger : TcLog;
END_VAR
TEST('LogsManyMessagesForManyCycles');

logsManyMessagesForManyCyclesLogger
  .WriteToFile('c:\UnitTest\', 'test.txt')
  .RunLogger();
logger.SetLogger(logsManyMessagesForManyCyclesLogger);

IF cycleCount < Cycles THEN
  FOR i:=0 TO Messages DO
    logger
      .AppendString('Cycle: ')
      .AppendString(UDINT_TO_STRING(cycleCount))
      .AppendString(', Message: ')
      .AppendString(UDINT_TO_STRING(i))
      .Error(''); 
  END_FOR
END_IF
cycleCount := cycleCount + 1;

// Catch any occuring error message
IF LEN(logsManyMessagesForManyCyclesLogger.Error.Info) > 0 THEN
  result := logsManyMessagesForManyCyclesLogger.Error.Info;
END_IF

IF cycleCount > (Cycles * Messages * 2 + 4) THEN 
  AssertEquals(Expected := expected,
         Actual := result,
         Message := result);
 
  TEST_FINISHED();
END_IF
END_METHOD

END_FUNCTION_BLOCK
